// Mitsubishi GX Works2 project: 신호등제어   PLC: Q03UDV

PROGRAM MAIN
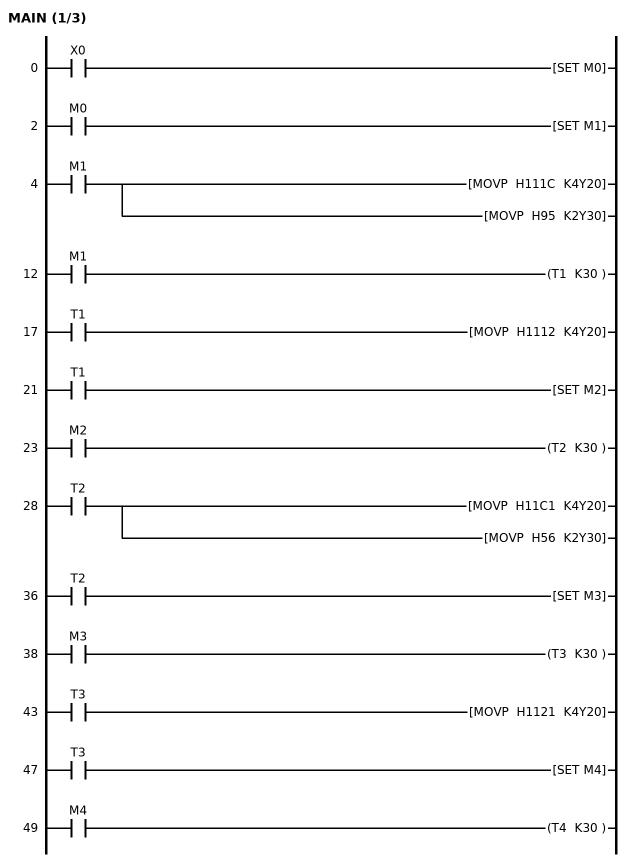
0     LD      X0
      SET     M0
2     LD      M0
      SET     M1
4     LD      M1
      MOVP    H111C K4Y20
      MOVP    H95 K2Y30
12    LD      M1
      OUT     T1 K30
17    LD      T1
      MOVP    H1112 K4Y20
21    LD      T1
      SET     M2
23    LD      M2
      OUT     T2 K30
28    LD      T2
      MOVP    H11C1 K4Y20
      MOVP    H56 K2Y30
36    LD      T2
      SET     M3
38    LD      M3
      OUT     T3 K30
43    LD      T3
      MOVP    H1121 K4Y20
47    LD      T3
      SET     M4
49    LD      M4
      OUT     T4 K30
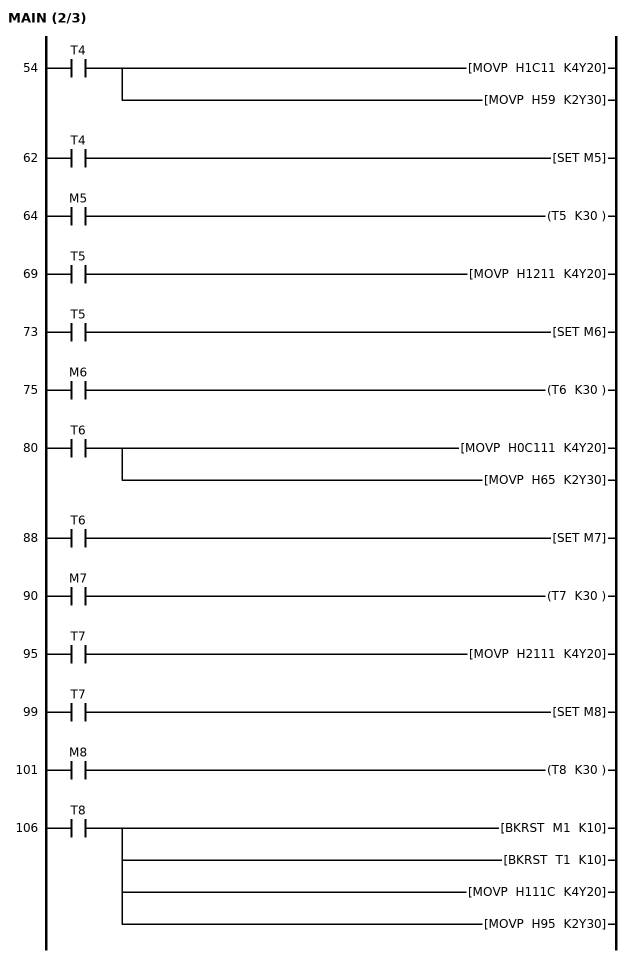
54    LD      T4
      MOVP    H1C11 K4Y20
      MOVP    H59 K2Y30
62    LD      T4
      SET     M5
64    LD      M5
      OUT     T5 K30
69    LD      T5
      MOVP    H1211 K4Y20
73    LD      T5
      SET     M6
75    LD      M6
      OUT     T6 K30
80    LD      T6
      MOVP    H0C111 K4Y20
      MOVP    H65 K2Y30
88    LD      T6
      SET     M7
90    LD      M7
      OUT     T7 K30
95    LD      T7
      MOVP    H2111 K4Y20
99    LD      T7
      SET     M8
101   LD      M8
      OUT     T8 K30
106   LD      T8
      BKRST   M1 K10
      BKRST   T1 K10
      MOVP    H111C K4Y20
      MOVP    H95 K2Y30
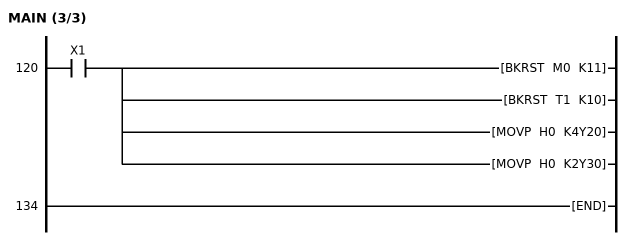
120   LD      X1
      BKRST   M0 K11
      BKRST   T1 K10
      MOVP    H0 K4Y20
      MOVP    H0 K2Y30
134   END
END_PROGRAM

PROGRAM MAIN1
0     END
END_PROGRAM
